Universal Robots PolyScope program: programa1-iniciales.urp

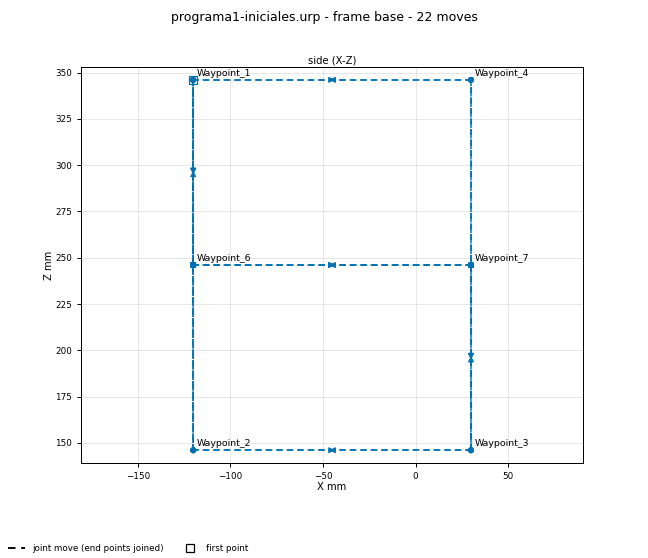
[picture p0: tool path of programa1-iniciales.urp in frame base, 22 of 22 moves have a stored position in this frame; points joined in program order, loops and branches not executed]
Program programa1- iniciales (installation=default directory=/ursim/programs createdIn=3.15.8.106339 lastSavedIn=3.15.8.106339 robotSerialNumber=2018359999)
Calibrated DH parameters: a=[0, -0.425, -0.39225, 0, 0, 0]; d=[0.089159, 0, 0, 0.10915, 0.09465, 0.0823]; alpha=[1.570796, 0, 0, 1.570796, -1.570796, 0]; deltaTheta=[0, 0, 0, 0, 0, 0]
Robot Program (runOnlyOnce=true)
  Popup Message (haltProgram=false message=Trayectoria de la letra L - Leydi Solorza  inputType=Text)
  MoveJ speed 60 deg/s, acceleration 80 deg/s^2 (useActiveTCP=true)
    Waypoint Waypoint_1: TCP in base x=-120.113 y=-431.763 z=346.07 mm, rx=-0.0012 ry=3.1163 rz=0.0389 rad; joints [-91.713, -84.457, -107.523, -79.493, 91.393, -1.776] deg
    Waypoint Waypoint_2: TCP in base x=-120.113 y=-431.763 z=146.073 mm, rx=-0.0012 ry=3.1163 rz=0.0389 rad; joints [-91.713, -98.956, -126.223, -46.295, 91.393, -1.776] deg
    Waypoint Waypoint_3: TCP in base x=29.89 y=-431.763 z=146.073 mm, rx=-0.0012 ry=3.1163 rz=0.0389 rad; joints [-71.788, -97.102, -128.67, -45.139, 91.811, 18.153] deg
  Popup Message (haltProgram=false message=Trayectoria de la letra S  inputType=Text)
  MoveJ speed 60 deg/s, acceleration 80 deg/s^2 (useActiveTCP=true)
    Waypoint Waypoint_4: TCP in base x=29.89 y=-431.763 z=346.07 mm, rx=-0.0012 ry=3.1163 rz=0.0389 rad; joints [-71.788, -82.186, -109.64, -79.084, 91.811, 18.153] deg
    Waypoint Waypoint_5: TCP in base x=-120.11 y=-431.763 z=346.07 mm, rx=-0.0012 ry=3.1163 rz=0.0389 rad; joints [-91.713, -84.457, -107.523, -79.493, 91.393, -1.776] deg
    Waypoint Waypoint_6: TCP in base x=-120.11 y=-431.763 z=246.07 mm, rx=-0.0012 ry=3.1163 rz=0.0389 rad; joints [-91.713, -89.449, -118.424, -63.599, 91.393, -1.776] deg
    Waypoint Waypoint_7: TCP in base x=29.89 y=-431.763 z=246.07 mm, rx=-0.0012 ry=3.1163 rz=0.0389 rad; joints [-71.788, -87.255, -120.695, -62.96, 91.811, 18.153] deg
    Waypoint Waypoint_8: TCP in base x=29.89 y=-431.763 z=146.07 mm, rx=-0.0012 ry=3.1163 rz=0.0389 rad; joints [-71.788, -97.102, -128.67, -45.138, 91.811, 18.153] deg
    Waypoint Waypoint_9: TCP in base x=-120.11 y=-431.763 z=146.07 mm, rx=-0.0012 ry=3.1163 rz=0.0389 rad; joints [-91.713, -98.956, -126.223, -46.294, 91.393, -1.776] deg
  Popup Message (haltProgram=false message=Trayectoria de la letra A - Alejandro Huertas inputType=Text)
  MoveJ speed 60 deg/s, acceleration 80 deg/s^2 (useActiveTCP=true)
    Waypoint Waypoint_10: TCP in base x=-120.11 y=-431.76 z=146.07 mm, rx=-0.0012 ry=3.1163 rz=0.0389 rad; joints [-91.713, -98.955, -126.223, -46.294, 91.393, -1.776] deg
    Waypoint Waypoint_11: TCP in base x=-120.11 y=-431.76 z=346.07 mm, rx=-0.0012 ry=3.1163 rz=0.0389 rad; joints [-91.713, -84.457, -107.523, -79.493, 91.393, -1.776] deg
    Waypoint Waypoint_12: TCP in base x=29.89 y=-431.76 z=346.07 mm, rx=-0.0012 ry=3.1163 rz=0.0389 rad; joints [-71.788, -82.186, -109.64, -79.084, 91.811, 18.153] deg
    Waypoint Waypoint_13: TCP in base x=29.89 y=-431.76 z=146.07 mm, rx=-0.0012 ry=3.1163 rz=0.0389 rad; joints [-71.788, -97.102, -128.671, -45.138, 91.811, 18.153] deg
    Waypoint Waypoint_14: TCP in base x=29.89 y=-431.76 z=246.07 mm, rx=-0.0012 ry=3.1163 rz=0.0389 rad; joints [-71.788, -87.255, -120.695, -62.96, 91.811, 18.153] deg
    Waypoint Waypoint_15: TCP in base x=-120.11 y=-431.76 z=246.07 mm, rx=-0.0012 ry=3.1163 rz=0.0389 rad; joints [-91.713, -89.449, -118.425, -63.599, 91.393, -1.776] deg
    Waypoint Waypoint_16: TCP in base x=-120.11 y=-431.76 z=346.07 mm, rx=-0.0012 ry=3.1163 rz=0.0389 rad; joints [-91.713, -84.457, -107.523, -79.493, 91.393, -1.776] deg
  Popup Message (haltProgram=false message=Trayectoria de la letra H  inputType=Text)
  MoveJ speed 60 deg/s, acceleration 80 deg/s^2 (useActiveTCP=true)
    Waypoint Waypoint_17: TCP in base x=-120.113 y=-431.763 z=146.073 mm, rx=-0.0012 ry=3.1163 rz=0.0389 rad; joints [-91.713, -98.956, -126.223, -46.295, 91.393, -1.776] deg
    Waypoint Waypoint_18: TCP in base x=-120.113 y=-431.763 z=346.07 mm, rx=-0.0012 ry=3.1163 rz=0.0389 rad; joints [-91.713, -84.457, -107.523, -79.493, 91.393, -1.776] deg
    Waypoint Waypoint_19: TCP in base x=-120.11 y=-431.763 z=246.07 mm, rx=-0.0012 ry=3.1163 rz=0.0389 rad; joints [-91.713, -89.449, -118.424, -63.599, 91.393, -1.776] deg
    Waypoint Waypoint_20: TCP in base x=29.89 y=-431.763 z=246.07 mm, rx=-0.0012 ry=3.1163 rz=0.0389 rad; joints [-71.788, -87.255, -120.695, -62.96, 91.811, 18.153] deg
    Waypoint Waypoint_21: TCP in base x=29.89 y=-431.763 z=146.07 mm, rx=-0.0012 ry=3.1163 rz=0.0389 rad; joints [-71.788, -97.102, -128.67, -45.138, 91.811, 18.153] deg
    Waypoint Waypoint_22: TCP in base x=29.89 y=-431.763 z=346.07 mm, rx=-0.0012 ry=3.1163 rz=0.0389 rad; joints [-71.788, -82.186, -109.64, -79.084, 91.811, 18.153] deg
